PROGRAM motor_starter_control_st
VAR PERSISTENT
	
END_VAR

END_PROGRAM

(* stored: Version 1.1.0.1, ProductVersion 3.1.4024.12
   POU motor_starter_control_st: Id {ef6ee357-7fc9-4352-87a7-88c91e076efb}, SpecialFunc None *)
